Fanuc KAREL source: kt00909.KL

-- PROVISIONAL review KL for V940-1; original PC SHA256 29781da7ed0b4d134317d9b2c5b8cf7169a96a52598b9dbc4fb0eed82dee3821
-- Incomplete behavior may be omitted. Consult companion uncertainty JSON. Do not deploy.
PROGRAM KT00909
%NOLOCKGROUP
BEGIN
  -- V9_ZERO_TABLE_METADATA_HINT layout=0002_ascii; no indexed target words; source/name/runtime held
  -- UNRESOLVED_PC offsets 5-20; opcodes 2E,22,32,35
  -- UNRESOLVED_PC offsets 25-40; opcodes 2E,22,32,35
  -- UNRESOLVED_PC offsets 45-60; opcodes 2E,22,32,35
  -- UNRESOLVED_PC offsets 65-80; opcodes 2E,22,32,35
  -- UNRESOLVED_PC offsets 85-111; opcodes 27,27,49,7E,AD,31,4A
  -- UNRESOLVED_PC offsets 116-120; opcodes 7F
END KT00909
